{attribute addProperty BoxType "EK1122-0000-0018"}
{attribute addProperty Id "Beckhoff_EL19xxsub_EK1100EK1100_179A0949162"}
{attribute addProperty CRC "3728394877"}
{attribute addProperty SizeInBites "16"}
{attribute addProperty SizeInBytes "2"}
TYPE Beckhoff_EL19xxEK1122_DE3ACA7D EXTENDS EK1122_179A0949 :
STRUCT
	{attribute addProperty Name "Beckhoff_EL19xxsub_EK1100"}
	Beckhoff_EL19xxsub_EK1100 : EK1100_179A0949;
END_STRUCT
END_TYPE

(* stored: Version 1.2.0.0, ProductVersion 3.1.4024.9
   DUT Beckhoff_EL19xxEK1122_DE3ACA7D: Id {a69d72ac-5f52-4160-83a3-5e978783e010} *)
